// TIA Portal V21 export
DATA_BLOCK "DispositivoProfinet"   // DB33
{ S7_Optimized_Access := 'TRUE' }
// stored: MemoryReserve 100
   VAR
      D : Array[0.."K_NumDispositivoProfinet"] of "Std_DispositivoProfinet";
   END_VAR
BEGIN
   D[0].Allarmi."A"[0..1].Abilitato := FALSE;
   D[0].Allarmi."A"[0..1].Stato := FALSE;
   D[0].Allarmi."A"[0..1].Silenziato := FALSE;
   D[0].Allarmi."A"[0..1].EnWarnHmi := FALSE;
   D[0].Allarmi."A"[0..1].EnCadutaCiclo := FALSE;
   D[0].Allarmi.WordHMI := 16#0000;
END_DATA_BLOCK
